TYPE ST_PROCESS_STATE :
STRUCT
  State           : E_PROCESS_STATE;
  Result          : E_PROGRESS;
  Check           : E_PROCESS_CHECK;
END_STRUCT
END_TYPE

(* stored: Version 1.1.0.1, ProductVersion 3.1.4024.13
   DUT ST_PROCESS_STATE: Id {44610655-ffe8-45f1-96ce-a5b382121307} *)
